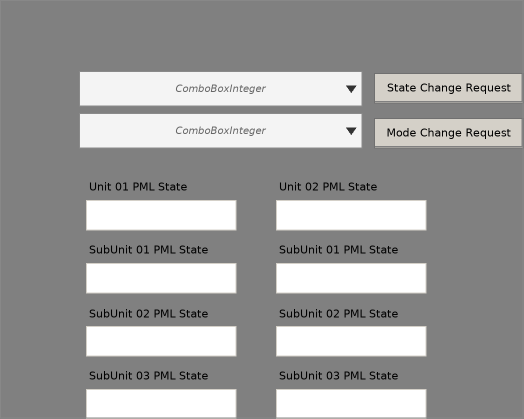
VISUALIZATION Visualization  // 524x419
    ComboBoxInteger (79,71 283x35), variable: GVL.LineCommands.Command.CntrlCmd, text list: 'tlPML_Commands'
    Button (374,118 150x30), "Mode Change Request"
        tap GVL.UnitPackTags[2].Command.UnitModeChangeRequest
    ComboBoxInteger (79,113 283x35), variable: GVL.LineCommands.Command.UnitMode, text list: 'tlPML_Modes'
    Button (374,73 150x30), "State Change Request"
        tap GVL.LineCommands.Command.CmdChangeRequest
    Textfield (86,200 150x30), text list: 'tlPML_States', text index: PackML_01.fbRobotCell.eState
    Label (86,172 149x30), "Unit 01 PML State"
    Textfield (86,263 150x30), text list: 'tlPML_States', text index: PackML_01.fbInfeed.eState
    Label (86,235 149x30), "SubUnit 01 PML State"
    Textfield (86,326 150x30), text list: 'tlPML_States', text index: PackML_01.fbDelta.eState
    Label (86,299 149x30), "SubUnit 02 PML State"
    Textfield (86,389 150x30), text list: 'tlPML_States', text index: PackML_01.fbDischarge.eState
    Label (86,361 149x30), "SubUnit 03 PML State"
    Textfield (276,200 150x30), text list: 'tlPML_States', text index: PackML_02.fbRobotCell.eState
    Label (276,172 149x30), "Unit 02 PML State"
    Textfield (276,263 150x30), text list: 'tlPML_States', text index: PackML_02.fbInfeed.eState
    Label (276,235 149x30), "SubUnit 01 PML State"
    Textfield (276,326 150x30), text list: 'tlPML_States', text index: PackML_02.fbScara.eState
    Label (276,299 149x30), "SubUnit 02 PML State"
    Textfield (276,389 150x30), text list: 'tlPML_States', text index: PackML_02.fbDischarge.eState
    Label (276,361 149x30), "SubUnit 03 PML State"
END_VISUALIZATION

(* stored: Version 1.1.0.1, ProductVersion 3.1.4024.11
   Visu Visualization: Id {61be7c6c-cc14-4139-8a67-351b42ef3e8c} *)
